// Tests for AstroBROT.FB_SUNPOS (apparent position of the Sun, port of IDLAstro sunpos.pro).
//
// GENERATED by AstroBROT/testing/gen_block_tests.py from testing/golden_blocks.py, do not edit the numbers by hand.
// Golden values from the Python port of the ST (1E-7 deg). Independently of the port the position is compared with a
// position built from erfa (epv00 / pmat06 / nut06a): 1.5E-3 deg = 5.4 arcsec, the measured maximum is 3.2 arcsec and
// the IDLAstro documentation states 7.3 arcsec for 1900-2100. The last tests are plain sanity checks (equinox,
// solstice, obliquity, RA rate) that need neither the port nor erfa.
FUNCTION_BLOCK FB_SUNPOS_Tests EXTENDS TcUnit.FB_TestSuite
VAR
END_VAR

Golden_Epoch_1900_And_J2000();
Golden_Start_2010();
Golden_Tenerife_2026();
Golden_Year_2050();
Golden_Equinox_And_Solstice_2026();
Sanity_Equinox_Solstice_Obliquity();
Sanity_Right_Ascension_Advances_About_One_Degree_Per_Day();
Inputs_Are_Not_Modified();
Cyclic_Calls_With_Inputs_Set_Once_Are_Stable();

METHOD PRIVATE CheckNear
VAR_INPUT
	fExpected	: LREAL;
	fActual	: LREAL;
	fDelta	: LREAL;
	sName	: STRING(255);
END_VAR
AssertEquals_LREAL(Expected := fExpected, Actual := fActual, Delta := fDelta, Message := sName);
END_METHOD

METHOD PRIVATE CheckAngle
VAR_INPUT
	fExpected	: LREAL;
	fActual	: LREAL;
	fDelta	: LREAL;
	sName	: STRING(255);
END_VAR
VAR
	fDiff	: LREAL;
END_VAR
// angles in degrees, compared modulo 360 so that 359.9999999 and -1.0E-7 are equal
fDiff := fActual - fExpected;
WHILE fDiff > 180.0 DO fDiff := fDiff - 360.0; END_WHILE
WHILE fDiff < -180.0 DO fDiff := fDiff + 360.0; END_WHILE
AssertEquals_LREAL(Expected := 0.0, Actual := fDiff, Delta := fDelta, Message := sName);
END_METHOD

METHOD PRIVATE CheckSeparation
VAR_INPUT
	fLon1	: LREAL;
	fLat1	: LREAL;
	fLon2	: LREAL;
	fLat2	: LREAL;
	fDelta	: LREAL;
	sName	: STRING(255);
END_VAR
VAR
	fD2r	: LREAL;
	fHalfDLat	: LREAL;
	fHalfDLon	: LREAL;
	fHav	: LREAL;
	fSep	: LREAL;
END_VAR
// great-circle separation of two positions (longitude, latitude in degrees) against a tolerance in degrees;
// a difference of longitudes is not a distance on the sky, this is (haversine formula)
fD2r := 0.017453292519943295;
fHalfDLat := (fLat2 - fLat1) * fD2r * 0.5;
fHalfDLon := (fLon2 - fLon1) * fD2r * 0.5;
fHav := SIN(fHalfDLat) * SIN(fHalfDLat) + COS(fLat1 * fD2r) * COS(fLat2 * fD2r) * SIN(fHalfDLon) * SIN(fHalfDLon);
fSep := 2.0 * ASIN(SQRT(LIMIT(0.0, fHav, 1.0))) / fD2r;
AssertEquals_LREAL(Expected := 0.0, Actual := fSep, Delta := fDelta, Message := sName);
END_METHOD

METHOD PRIVATE Golden_Epoch_1900_And_J2000
VAR
	fb	: AstroBROT.FB_SUNPOS;
END_VAR
TEST('Golden_Epoch_1900_And_J2000');
fb(jd := 2415020.0);
CheckAngle(280.4932027906667, fb.ra, 1.0E-7, 'Epoch_1900 ra');
CheckNear(-23.1010537507843, fb.dec, 1.0E-7, 'Epoch_1900 dec');
CheckNear(279.6444003923051, fb.longmed, 1.0E-7, 'Epoch_1900 longmed');
CheckNear(23.451814403891508, fb.oblt, 1.0E-7, 'Epoch_1900 oblt');
CheckSeparation(280.49336588705194, -23.100882447052207, fb.ra, fb.dec, 0.0015, 'Epoch_1900 vs erfa');
fb(jd := 2451545.0);
CheckAngle(281.27675114506104, fb.ra, 1.0E-7, 'J2000 ra');
CheckNear(-23.03291144063576, fb.dec, 1.0E-7, 'J2000 dec');
CheckNear(280.37698786565545, fb.longmed, 1.0E-7, 'J2000 longmed');
CheckNear(23.437814186179185, fb.oblt, 1.0E-7, 'J2000 oblt');
CheckSeparation(281.2776898567173, -23.032708521099703, fb.ra, fb.dec, 0.0015, 'J2000 vs erfa');
TEST_FINISHED();
END_METHOD

METHOD PRIVATE Golden_Start_2010
VAR
	fb	: AstroBROT.FB_SUNPOS;
END_VAR
TEST('Golden_Start_2010');
fb(jd := 2455197.5);
CheckAngle(281.36670259981736, fb.ra, 1.0E-7, 'Start_2010 ra');
CheckNear(-23.027520406003863, fb.dec, 1.0E-7, 'Start_2010 dec');
CheckNear(280.4515850797381, fb.longmed, 1.0E-7, 'Start_2010 longmed');
CheckNear(23.438922135094707, fb.oblt, 1.0E-7, 'Start_2010 oblt');
CheckSeparation(281.3668435021951, -23.027353107638568, fb.ra, fb.dec, 0.0015, 'Start_2010 vs erfa');
TEST_FINISHED();
END_METHOD

METHOD PRIVATE Golden_Tenerife_2026
VAR
	fb	: AstroBROT.FB_SUNPOS;
END_VAR
TEST('Golden_Tenerife_2026');
fb(jd := 2461300.75);
CheckAngle(174.8393337772982, fb.ra, 1.0E-7, 'Tenerife_2026 ra');
CheckNear(2.2331274030840897, fb.dec, 1.0E-7, 'Tenerife_2026 dec');
CheckNear(174.38128640738705, fb.longmed, 1.0E-7, 'Tenerife_2026 longmed');
CheckNear(23.437983366242445, fb.oblt, 1.0E-7, 'Tenerife_2026 oblt');
CheckSeparation(174.84005201634432, 2.232830546071217, fb.ra, fb.dec, 0.0015, 'Tenerife_2026 vs erfa');
TEST_FINISHED();
END_METHOD

METHOD PRIVATE Golden_Year_2050
VAR
	fb	: AstroBROT.FB_SUNPOS;
END_VAR
TEST('Golden_Year_2050');
fb(jd := 2469807.5);
CheckAngle(281.68738605381645, fb.ra, 1.0E-7, 'Year_2050 ra');
CheckNear(-22.996590225692305, fb.dec, 1.0E-7, 'Year_2050 dec');
CheckNear(280.748664812077, fb.longmed, 1.0E-7, 'Year_2050 longmed');
CheckNear(23.431419887249728, fb.oblt, 1.0E-7, 'Year_2050 oblt');
CheckSeparation(281.6880601925095, -22.996415910571415, fb.ra, fb.dec, 0.0015, 'Year_2050 vs erfa');
TEST_FINISHED();
END_METHOD

METHOD PRIVATE Golden_Equinox_And_Solstice_2026
VAR
	fb	: AstroBROT.FB_SUNPOS;
END_VAR
TEST('Golden_Equinox_And_Solstice_2026');
fb(jd := 2461120.5);
CheckAngle(0.3503559250411667, fb.ra, 1.0E-7, 'March_equinox_2026 ra');
CheckNear(0.15188894029624206, fb.dec, 1.0E-7, 'March_equinox_2026 dec');
CheckNear(0.3857660381664108, fb.longmed, 1.0E-7, 'March_equinox_2026 longmed');
CheckNear(23.438239257244735, fb.oblt, 1.0E-7, 'March_equinox_2026 oblt');
CheckSeparation(0.35013805050580776, 0.15179565874940165, fb.ra, fb.dec, 0.0015, 'March_equinox_2026 vs erfa');
fb(jd := 2461212.5);
CheckAngle(89.63389115907498, fb.ra, 1.0E-7, 'June_solstice_2026 ra');
CheckNear(23.437689690338015, fb.dec, 1.0E-7, 'June_solstice_2026 dec');
CheckNear(89.66763149502222, fb.longmed, 1.0E-7, 'June_solstice_2026 longmed');
CheckNear(23.43811655330089, fb.oblt, 1.0E-7, 'June_solstice_2026 oblt');
CheckSeparation(89.63460394632473, 23.437550528896672, fb.ra, fb.dec, 0.0015, 'June_solstice_2026 vs erfa');
TEST_FINISHED();
END_METHOD

METHOD PRIVATE Sanity_Equinox_Solstice_Obliquity
VAR
	fb	: AstroBROT.FB_SUNPOS;
END_VAR
TEST('Sanity_Equinox_Solstice_Obliquity');
// 2026-03-21 00:00 UT is 9 h after the March equinox: the Sun is at RA about 0.35 deg, Dec about +0.15 deg
fb(jd := 2461120.5);
CheckAngle(0.35, fb.ra, 0.3, 'March equinox ra');
CheckNear(0.15, fb.dec, 0.1, 'March equinox dec');
// 2026-06-21 00:00 UT is 8 h before the June solstice: Dec is at its maximum, RA about 89.6 deg
fb(jd := 2461212.5);
CheckNear(23.44, fb.dec, 0.02, 'June solstice dec');
CheckAngle(89.6, fb.ra, 0.3, 'June solstice ra');
// true obliquity of the ecliptic in 2026
CheckNear(23.437, fb.oblt, 0.005, 'oblt 2026');
TEST_FINISHED();
END_METHOD

METHOD PRIVATE Sanity_Right_Ascension_Advances_About_One_Degree_Per_Day
VAR
	fb	: AstroBROT.FB_SUNPOS;
	fbNext	: AstroBROT.FB_SUNPOS;
	i	: INT;
	fStep	: LREAL;
END_VAR
TEST('Sanity_Right_Ascension_Advances_About_One_Degree_Per_Day');
// over a year the daily change of RA is between 0.85 and 1.15 deg (0.91 to 1.11 in reality); this also crosses the wrap at 360
FOR i := 0 TO 36 DO
	fb(jd := 2461041.5 + 10.0 * i);
	fbNext(jd := 2461042.5 + 10.0 * i);
	fStep := fbNext.ra - fb.ra;
	IF fStep < 0.0 THEN fStep := fStep + 360.0; END_IF
	AssertTrue(Condition := fStep > 0.85 AND fStep < 1.15, Message := 'daily RA step within 0.85 .. 1.15 deg');
	AssertTrue(Condition := fb.ra >= 0.0 AND fb.ra < 360.0 AND ABS(fb.dec) < 23.5, Message := 'ra in range, |dec| below the obliquity');
END_FOR
TEST_FINISHED();
END_METHOD

METHOD PRIVATE Inputs_Are_Not_Modified
VAR
	fb	: AstroBROT.FB_SUNPOS;
END_VAR
TEST('Inputs_Are_Not_Modified');
fb(jd := 2461300.75);
CheckNear(2461300.75, fb.jd, 0.0, 'jd unchanged');
TEST_FINISHED();
END_METHOD

METHOD PRIVATE Cyclic_Calls_With_Inputs_Set_Once_Are_Stable
VAR
	fb	: AstroBROT.FB_SUNPOS;
	i	: INT;
END_VAR
TEST('Cyclic_Calls_With_Inputs_Set_Once_Are_Stable');
fb.jd := 2461300.75;
FOR i := 1 TO 5 DO
	fb();
	CheckAngle(174.8393337772982, fb.ra, 1.0E-7, 'cyclic call ra');
	CheckNear(2.2331274030840897, fb.dec, 1.0E-7, 'cyclic call dec');
END_FOR
TEST_FINISHED();
END_METHOD

END_FUNCTION_BLOCK

(* stored: Version 1.1.0.1, ProductVersion 3.1.4024.15
   POU FB_SUNPOS_Tests: Id {0f6f9c9c-5d39-544c-a01d-cfbc113d5682}, SpecialFunc None
   Method CheckNear: Id {f01afbd0-b4fb-5cbd-856f-a3ba23664208}
   Method CheckAngle: Id {b1726c49-0452-559e-993a-3347036f4177}
   Method CheckSeparation: Id {ffe23ca7-02a1-542b-8e1b-ae6d45ac189c}
   Method Golden_Epoch_1900_And_J2000: Id {b57dcbde-72a8-5f87-9202-17d98d926790}
   Method Golden_Start_2010: Id {4fb8541c-eeef-55f0-b460-58e3d0c43126}
   Method Golden_Tenerife_2026: Id {ecac9414-5511-536d-a6d2-9c35c54cd843}
   Method Golden_Year_2050: Id {5133d389-04d6-5400-aed8-eb12daa80383}
   Method Golden_Equinox_And_Solstice_2026: Id {96178e92-4e92-57e4-8dd7-913f9b338974}
   Method Sanity_Equinox_Solstice_Obliquity: Id {11c5d72b-7ff4-509c-a04f-41e2a68a7249}
   Method Sanity_Right_Ascension_Advances_About_One_Degree_Per_Day: Id {c3440e0f-4170-5c24-a36f-cd561b32813a}
   Method Inputs_Are_Not_Modified: Id {33f65d12-80f6-5ee1-8fb7-9afeab0a7580}
   Method Cyclic_Calls_With_Inputs_Set_Once_Are_Stable: Id {3be82c5d-3cef-53f3-a617-a182a53e24a5} *)
